// TIA Portal V18 export
// export: Created 2025-12-01T17:51:23.2597848Z, ExportSetting None, DisplayName Totally Integrated Automation Portal, DisplayVersion V18 Update 5, DisplayName TIA Portal Openness, DisplayVersion V18 Update 5, DisplayName TIA Portal Teamcenter Gateway, DisplayVersion V18, DisplayName TIA Portal Version Control Interface, DisplayVersion V18, DisplayName STEP 7 Professional, DisplayVersion V18 Update 5, DisplayName STEP 7 Safety, DisplayVersion V18, DisplayName WinCC Professional, DisplayVersion V18 Update 5
DATA_BLOCK "ST10_PLC_GetDB"   // DB901
{ S7_Optimized_Access := 'FALSE' }
// stored: AutoNumber false
   VAR
      InData : Struct
         Global : Struct
            Beat : Bool;
            AutoRunning : Bool;
            Alarm : Bool;
            SystemStandby : Bool;
            AutoMode : Bool;
            ManualMode : Bool;
            Spare_4 : Bool;
            Spare_5 : Bool;
            Spare_6 : Bool;
            Spare_7 : Bool;
            Spare_8 : Bool;
            Spare_9 : Bool;
            Spare_10 : Bool;
            Spare_11 : Bool;
            Spare_12 : Bool;
            Spare_13 : Bool;
         END_STRUCT;
         Control : Struct
            AskPallet : Bool;
            PalletInPos : Bool;
            Spare_1 : Bool;
            Spare_2 : Bool;
            Spare_3 : Bool;
            Spare_4 : Bool;
            Spare_5 : Bool;
            Spare_6 : Bool;
            Spare_7 : Bool;
            Spare_8 : Bool;
            Spare_9 : Bool;
            Spare_10 : Bool;
            Spare_11 : Bool;
            Spare_12 : Bool;
            Spare_13 : Bool;
            Spare_14 : Byte;
            Spare_15 : Byte;
         END_STRUCT;
         Data : Struct
            CurrentTemperature_1 : Int;
            CurrentTemperature_2 : Int;
            SetTemperature : Int;
            SetSolidifyTime : Int;
            ActualSolidifyTime : Int;   // Min
            Spare_3 : Array[0..83] of Byte;
         END_STRUCT;
      END_STRUCT;
   END_VAR
BEGIN
END_DATA_BLOCK
